PROGRAM MAIN
VAR
END_VAR

END_PROGRAM

(* stored: Version 1.1.0.1
   POU MAIN: Id {22afe78e-d291-4978-8f1c-44f9db8c72fa} *)
